TYPE ST_OvercurrentProtection_InternalLinking :
STRUCT
	a_r_CurrentInput			: ARRAY [1..2] OF ARRAY[1..4] OF REAL; //first array of powerlockset, second of powerlock
	a_r_CurrentOutput			: ARRAY [1..3] OF ARRAY[1..4] OF REAL;
	b_InputSectionAvailable 	: BOOL;
	b_thirdOutputAvailable 		: BOOL;
END_STRUCT
END_TYPE

(* stored: Version 1.1.0.1, ProductVersion 3.1.4026.18
   DUT ST_OvercurrentProtection_InternalLinking: Id {b0e61979-3fdc-433c-8b9e-591250c843bb} *)
